INTERFACE IReadOnlyList EXTENDS ICollection

METHOD FindSingle : BOOL
VAR_INPUT
	predicate : IPredicate;
	skip : UDINT := 0;
	searchDirection : SEARCH_DIRECTION := SEARCH_DIRECTION.FROM_BEGINNING;
END_VAR
VAR_OUTPUT
	value : GENERIC_VALUE;
	index : DINT;
END_VAR
END_METHOD

METHOD Get : REFERENCE TO GENERIC_VALUE
VAR_INPUT
	index : DINT;
END_VAR
END_METHOD

END_INTERFACE

(* stored: Version 1.1.0.1
   Itf IReadOnlyList: Id {2ae0731d-8d43-42f2-abee-f0660bf607da}
   Method FindSingle: Id {1b102e63-f5bc-45b5-87cf-c33b4c4088e7}
   Method Get: Id {f5cd9212-1ade-4b6f-92a1-97d3e216a850} *)
